// Implicitly generated code : DO NOT EDIT
FUNCTION CheckLRangeSigned : LINT
VAR_INPUT
	value, lower, upper: LINT;
END_VAR
VAR
    sMessageLow   : STRING := 'CheckLRangeSigned: Value too low (%d)';
    sMessageHigh  : STRING := 'CheckLRangeSigned: Value too high (%d)';
END_VAR

// Implicitly generated code : Only an Implementation suggestion
{noflow}
IF (value < lower) THEN
	CheckLRangeSigned := lower;
	// Log message
    ADSLOGLREAL(msgCtrlMask := ADSLOG_MSGTYPE_WARN,
               msgFmtStr   := sMessageLow,
               lrealArg     := TO_REAL(value));
ELSIF(value > upper) THEN
	CheckLRangeSigned := upper;
	// Log message
    ADSLOGLREAL(msgCtrlMask := ADSLOG_MSGTYPE_WARN,
               msgFmtStr   := sMessageHigh,
               lrealArg     := TO_REAL(value));
ELSE
	CheckLRangeSigned := value;
END_IF

{flow}

END_FUNCTION

(* stored: Version 1.1.0.1, ProductVersion 3.1.4024.11
   POU CheckLRangeSigned: Id {c3d26626-36aa-401e-998e-9202de1182f8}, SpecialFunc CheckLRangeSigned *)
